Fanuc TP program (LS listing): shipping.ls

/PROG  SHIPPING
/ATTR
OWNER		= MNEDITOR;
COMMENT		= "";
PROG_SIZE	= 480;
CREATE		= DATE 25-08-25  TIME 12:54:04;
MODIFIED	= DATE 25-08-25  TIME 12:54:18;
FILE_NAME	= ;
VERSION		= 0;
LINE_COUNT	= 1;
MEMORY_SIZE	= 848;
PROTECT		= READ_WRITE;
TCD:  STACK_SIZE	= 0,
      TASK_PRIORITY	= 50,
      TIME_SLICE	= 0,
      BUSY_LAMP_OFF	= 0,
      ABORT_REQUEST	= 0,
      PAUSE_REQUEST	= 0;
DEFAULT_GROUP	= 1,*,*,*,*;
CONTROL_CODE	= 00000000 00000000;
LOCAL_REGISTERS	= 0,0,0;
/APPL

AUTO_SINGULARITY_HEADER;
  ENABLE_SINGULARITY_AVOIDANCE   : TRUE;
/MN
   1:J P[1] 100% FINE    ;
/POS
P[1]{
   GP1:
	UF : 0, UT : 1,
	J1=   -30.000 deg,	J2=   -30.000 deg,	J3=   -50.000 deg,
	J4=     0.000 deg,	J5=   -40.000 deg,	J6=     0.000 deg
};
/END
